{attribute 'pack_mode' := '1'}
TYPE TRunDataLift :
STRUCT
	eLiftPos			: TLiftPos;
END_STRUCT
END_TYPE

(* stored: Version 1.1.0.1, ProductVersion 3.1.4022.12
   DUT TRunDataLift: Id {f9e4e119-e518-450d-8713-24cd8ad9691c} *)
